// LS Electric XG5000 project: 8_23
// PLC LSPLC
// module base 0 slot 0: 입출력 모듈:XBC-DR14E (DC 24V 입력 8점, 릴레이 출력 6점)

PROGRAM NewProgram (task: 스캔 프로그램)

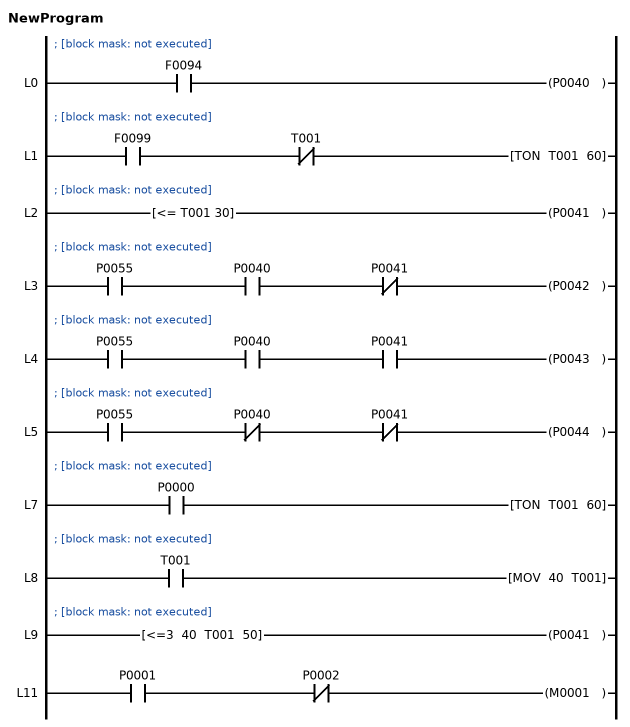
; L0 (block mask: not executed)
LOAD      F0094
OUT       P0040
; L1 (block mask: not executed)
LOAD      F0099
AND NOT   T001
TON       T001 60
; L2 (block mask: not executed)
LOAD<=    T001 30
OUT       P0041
; L3 (block mask: not executed)
LOAD      P0055
AND       P0040
AND NOT   P0041
OUT       P0042
; L4 (block mask: not executed)
LOAD      P0055
AND       P0040
AND       P0041
OUT       P0043
; L5 (block mask: not executed)
LOAD      P0055
AND NOT   P0040
AND NOT   P0041
OUT       P0044
; L7 (block mask: not executed)
LOAD      P0000
TON       T001 60
; L8 (block mask: not executed)
LOAD      T001
MOV       40 T001
; L9 (block mask: not executed)
LOAD<=3   40 T001 50
OUT       P0041
; L11
LOAD      P0001
AND NOT   P0002
OUT       M0001